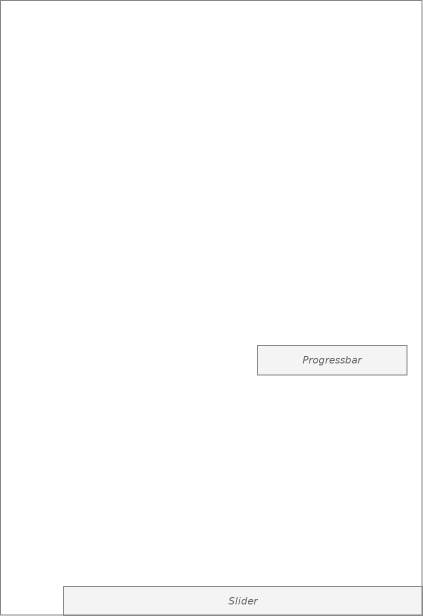
VISUALIZATION Visu  // 423x616
    Slider (63,586 360x30), variable: MAIN.nPmeter, scale 0..32767
    Progressbar (257,345 150x30), variable: MAIN.nValue
END_VISUALIZATION

(* stored: Version 1.1.0.1, ProductVersion 3.1.4024.12
   Visu Visu: Id {6760aef6-056a-4480-9dea-550790541f5f} *)
